{attribute 'qualified_only'}
VAR_GLOBAL
	fbFaultHandler : FB_FaultHandler; // The one and only faulthandler (a singleton)

	fbLogger : FB_LogToDisk(
					sLogFolder := PAR_Utilities.LOG_FOLDER,
					sLogFilePrefix := 'Log_',
					sLogFileExtension := 'txt',
					nMaxLogFileSize := 512*1024, // 512kb
					nMaxNumberOfLogFiles := 10
				);
END_VAR

(* stored: Version 1.1.0.1, ProductVersion 3.1.4024.11
   GVL GVL_Utilities: Id {6a3e625e-3b94-0b9e-27a1-84c13910a121} *)
